FUNCTION_BLOCK FB_IntervalBit
VAR_INPUT
	m_Input		: BOOL;			// Input which triggers the outputs accordingly
	t_Interval  : TIME;			// Time between the intervals 10s < Time < 12h
	t_HighTime	: TIME;			// Time for how long the output is high 100ms < Time < 5m
END_VAR
VAR_OUTPUT
	m_RisingEdge	: BOOL;		// Output shows the rising edge of the input (for t_HighTime)
	m_Interval		: BOOL;		// Output high when input high (for t_HighTime) and after t_Intervall (for t_HighTime) until input is low
	m_FallingEdge	: BOOL;		// Output shows the falling edge of the input (for t_HighTime)
END_VAR
VAR
	{attribute 'hide'}
	R_TRIG_0: r_trig;
	{attribute 'hide'}
	TP_0: tp;
	{attribute 'hide'}
	F_TRIG_0: f_trig;
	{attribute 'hide'}
	TP_1: tp;
	{attribute 'hide'}
	TP_2: tp;
	{attribute 'hide'}
	TON_0: ton;
END_VAR

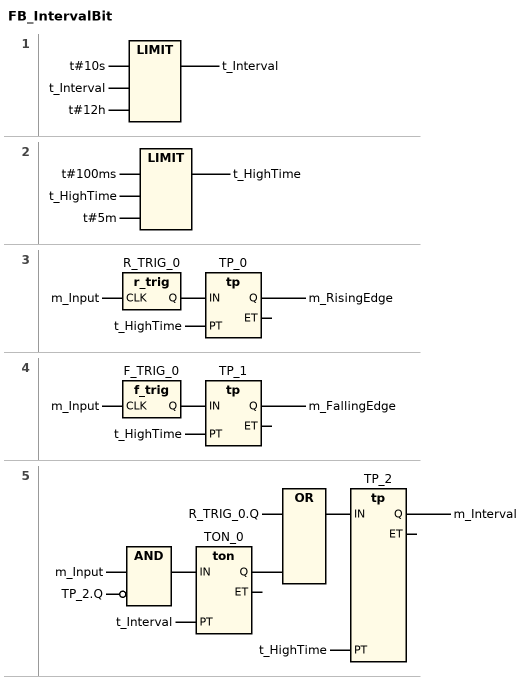
// NETWORK 1
t_Interval := LIMIT(t#10s, t_Interval, t#12h);

// NETWORK 2
t_HighTime := LIMIT(t#100ms, t_HighTime, t#5m);

// NETWORK 3
R_TRIG_0(CLK := m_Input); // r_trig
TP_0(IN := R_TRIG_0.Q, PT := t_HighTime); // tp
m_RisingEdge := TP_0.Q;

// NETWORK 4
F_TRIG_0(CLK := m_Input); // f_trig
TP_1(IN := F_TRIG_0.Q, PT := t_HighTime); // tp
m_FallingEdge := TP_1.Q;

// NETWORK 5
TON_0(IN := m_Input AND NOT TP_2.Q, PT := t_Interval); // ton
TP_2(IN := R_TRIG_0.Q OR TON_0.Q, PT := t_HighTime); // tp
m_Interval := TP_2.Q;

END_FUNCTION_BLOCK

(* stored: Version 1.1.0.1, ProductVersion 3.1.4024.12
   POU FB_IntervalBit: Id {2c71a4ef-806b-46a2-87f9-f5d14d8377e0}, SpecialFunc None *)
